// Implicitly generated code : DO NOT EDIT
FUNCTION CheckDivLReal : LREAL
VAR_INPUT
	divisor:LREAL;
END_VAR

// Implicitly generated code : Only an Implementation suggestion
IF divisor = 0 THEN
	CheckDivLReal:=1;
	nCheckDivLReal := nCheckDivLReal + 1;
ELSE
	CheckDivLReal:=divisor;
END_IF;

END_FUNCTION

(* stored: Version 1.1.0.1
   POU CheckDivLReal: Id {16fc3392-2ccc-412c-9989-821cbb04185d}, SpecialFunc CheckDivReal64 *)
